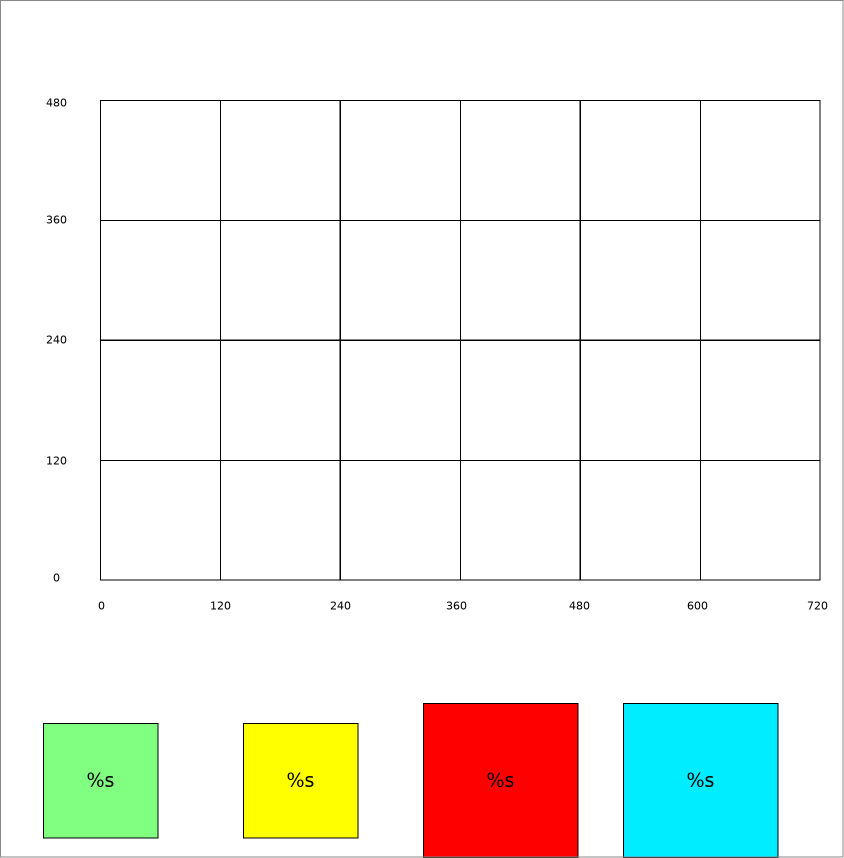
VISUALIZATION Visualization  // 844x858
    Label (75,588 53x36), "0"
    Label (194,588 53x36), "120"
    Label (314,588 53x36), "240"
    Label (430,588 53x36), "360"
    Label (553,588 53x36), "480"
    Label (671,588 53x36), "600"
    Label (791,588 53x36), "720"
    Rectangle (100,100 240x240)
    Rectangle (340,100 240x240)
    Rectangle (580,100 240x240)
    Rectangle (100,340 240x240)
    Rectangle (340,340 240x240)
    Rectangle (580,340 240x240)
    RoundedRectangle (423,703 155x155), "%s", text variable: Visu_Variable.strMoverText[3]
        p3560616238: Visu_Variable.stMoverPos[3].x
        p2738717112: Visu_Variable.stMoverPos[3].y
        p2277200375: Visu_Variable.stMoverPos[3].c
    RoundedRectangle (623,703 155x155), "%s", text variable: Visu_Variable.strMoverText[4]
        p3560616238: Visu_Variable.stMoverPos[4].x
        p2738717112: Visu_Variable.stMoverPos[4].y
        p2277200375: Visu_Variable.stMoverPos[4].c
    RoundedRectangle (43,723 115x115), "%s", text variable: Visu_Variable.strMoverText[1]
        p3560616238: Visu_Variable.stMoverPos[1].x
        p2738717112: Visu_Variable.stMoverPos[1].y
        p2277200375: Visu_Variable.stMoverPos[1].c
    RoundedRectangle (243,723 115x115), "%s", text variable: Visu_Variable.strMoverText[2]
        p3560616238: Visu_Variable.stMoverPos[2].x
        p2738717112: Visu_Variable.stMoverPos[2].y
        p2277200375: Visu_Variable.stMoverPos[2].c
    Line (220,100) (220,580)
    Line (460,100) (460,580)
    Line (700,100) (700,580)
    Line (100,220) (820,220)
    Line (100,460) (820,460)
    Label (30,560 53x36), "0"
    Label (30,443 53x36), "120"
    Label (30,322 53x36), "240"
    Label (30,202 53x36), "360"
    Label (30,85 53x36), "480"
END_VISUALIZATION

(* stored: Version 1.1.0.1, ProductVersion 3.1.4024.12
   Visu Visualization: Id {2449708a-7f90-4089-826a-75343f9c1bbf} *)
